RoboDK station: RoboDK.rdk

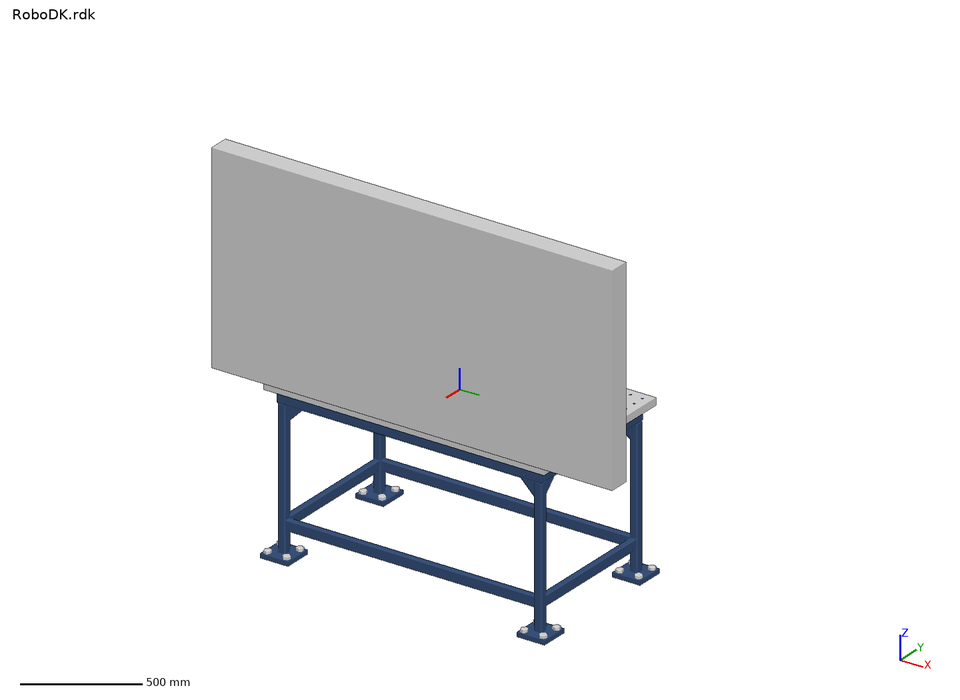
[picture v0: the station drawn from its stored meshes, robots at their saved joint values, targets as dots, program paths as lines]
Station Robotic (saved by RoboDK 5.6.8). Poses are relative to the parent item; angles as X-Y-Z fixed-axis rotations.
  - frame Mitsubishi RV-7FR Base at (0, 0, 0) mm, rotated rx 0 ry 0 rz -90 deg
    - robot Mitsubishi RV-7FR: 6 axes, payload 7 kg, reach 713 mm, repeatability 0.02 mm, weight 65 kg
        modified DH rows (alpha deg, a mm, theta deg, d mm): 0, 0, 0, 400; -90, 0, -90, 0; 0, 340, -90, 0; -90, 50, 0, 370; 90, 0, 0, 0; -90, 0, 180, 85
        joint limits [-240, -115, 0, -200, -120, -360] to [240, 125, 156, 200, 120, 360]; home [0, 0, 90, 0, 0, 0]; saved at [15.58, 20.58, 85.99, -28.57, -3.9, 35.06]
      - tool Sharpie v1, TCP at (0, 0, 150) mm, size 12.2 x 12.2 x 123.6 mm, geometry from Sharpie v1.stl
  - object Station Table at (-400, 0, 0) mm, size 1420 x 820 x 800 mm, geometry from Table.sld
  - Python program Prog1 (listed below)
  - object whiteboard v1 at (250, -700, 670) mm, rotated rx 0 ry 0 rz 90 deg, size 100 x 2000 x 1000 mm, geometry from whiteboard v1.stl

--- Python program Prog1 ---
#---------------------------------------------------
#--------------- PROGRAM START ---------------------
from robodk.robolink import * # API to communicate with RoboDK
from robodk.robomath import * # basic matrix operations
from robodk.robodialogs import *
from robodk.robofileio import *

RDK = Robolink()

# Generate the points curve path
#POINTS = MakePoints(P_START, P_END, NUM_POINTS)

# Ask the user to pick a file

# Input file name
#input_csv = getFileName(path_file) + ".csv"
input_csv = "C:\\Users\\nurbi\\Desktop\\abcPoint.csv"

# Output list to store the transformed data
output_data = []

# Read data from the input CSV file
with open(input_csv, 'r') as file:
    lines = file.readlines()

# Remove the header if it exists
header = lines.pop(0) if lines and ',' in lines[0] else None

# Process each line
output_data.append([500, float(lines[0].strip().split(',')[0])* -0.353 +600,
                    float(lines[0].strip().split(',')[1])* -0.353 +700])
for line in lines:
    if "#" in line:
        output_data.append([600, output_data[-1][1], output_data[-1][2]])
        continue

    # Assuming X is the first column and Y is the second column
    x, y = map(float, line.strip().split(','))

    # Convert X and Y to mm (multiply by 25.4)
    x_mm = -x * 0.353 +500
    y_mm = -y * 0.353 +700

    # Append a new row to the output data list
    output_data.append([600, x_mm, y_mm])

POINTS = output_data

# Initialize the RoboDK API
RDK = Robolink()

# turn off auto rendering (faster)
RDK.Render(False)

# Promt the user to select a robot (if only one robot is available
# it will select that robot automatically)
robot = RDK.ItemUserPick('Select a robot', ITEM_TYPE_ROBOT)

# Turn rendering ON before starting the simulation
RDK.Render(True)

# Abort if the user hits Cancel
if not robot.Valid():
    quit()

# Retrieve the robot reference frame
reference = robot.Parent()

# Use the robot base frame as the active reference
robot.setPoseFrame(reference)

# get the current orientation of the robot (with respect to the active
# reference frame and tool frame)
pose_ref = robot.Pose()
print(Pose_2_TxyzRxyz(pose_ref))

# a pose can also be defined as xyzwpr / xyzABC
#pose_ref = TxyzRxyz_2_Pose([100,200,300,0,0,pi])
#-------------------------------------------------------------
# Option 1: Move the robot using the Python script
# We can automatically force the "Create robot program" action usinga RUNMODE state
# RDK.setRunMode(RUNMODE_MAKE_ROBOTPROG)
# Iterate through all the points
for i in range(len(output_data)):
    # update the reference target with the desired XYZ coordinates
    pose_i = pose_ref
    pose_i.setPos(POINTS[i])
    # Move the robot to that target:
    robot.MoveJ(pose_i)
# Done, stop program execution
